(* Logix 5000 project; controller elevatorPart5 vendor 1 type 14 code 106 rev 28.11; software revision 28.03 *)

TASK MainTask (continuous, watchdog 500 ms) : MainProgram

MODULES
   Local : vendor 1 type 14 code 106 (Compact 0, rev 28.11)
       : vendor 1 type 7 code 77 (Compact 2, rev 3.1, Input RPI 20 ms)
       : 1769-IQ16 (Compact 3, rev 1.1, Input RPI 20 ms)
       : vendor 1 type 7 code 72 (Compact 5, rev 2.1, Output RPI 20 ms)
       : vendor 1 type 7 code 72 (Compact 4, rev 2.1, Output RPI 20 ms)
END_MODULES

ADD_ON_INSTRUCTION serviceDoor   (* revision 1.0 *)
VAR_OUTPUT
   serviceDoor : BOOL; {visible}
   doorOpen : BOOL; {visible}
   doorClosed : BOOL; {access Read Only, visible}
END_VAR
VAR_IN_OUT
   doorOpenSensor : BOOL; {required}
   doorClosedSensor : BOOL; {required}
END_VAR
VAR_OUTPUT
   doorControl : SINT; {access Read Only, visible}
END_VAR
VAR_IN_OUT
   pbOpenLyft : BOOL; {required}
   pbCloseLyft : BOOL; {required}
END_VAR
VAR
   doorOpenTimer : TIMER := (PRE := 5000); {access None}
   doorOpenTran : BOOL; {access None}
   activate : BOOL; {access None}
   lightOn : BOOL; {access None}
END_VAR

ROUTINE Logic   (* ladder *)
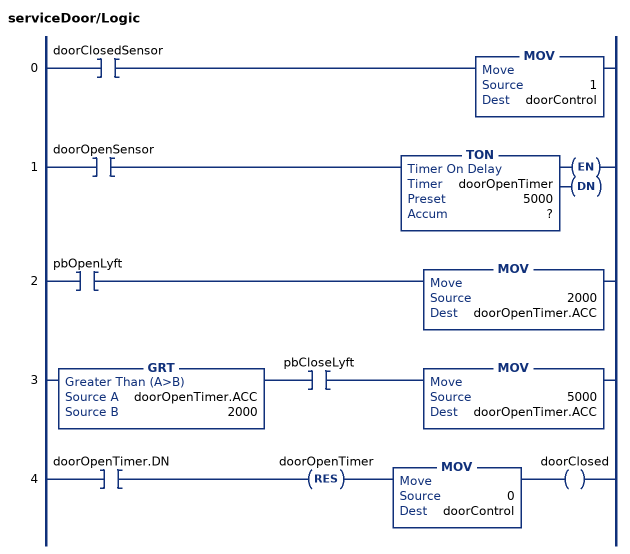
   0: XIC(doorClosedSensor)MOV(1,doorControl);
   1: XIC(doorOpenSensor)TON(doorOpenTimer,?,?);
   2: XIC(pbOpenLyft)MOV(2000,doorOpenTimer.ACC);
   3: GRT(doorOpenTimer.ACC,2000)XIC(pbCloseLyft)MOV(5000,doorOpenTimer.ACC);
   4: XIC(doorOpenTimer.DN)RES(doorOpenTimer)MOV(0,doorControl)OTE(doorClosed);
END_ROUTINE
END_ADD_ON_INSTRUCTION

PROGRAM MainProgram   (* main routine MainRoutine *)
VAR
   array : DINT[6];
   bits : DINT := 3855;
   bool : serviceDoor; {access Read Only}
   buttonPressDetection : SINT;
   callAddOn : BOOL;
   clearCount : DINT;
   count : DINT := 6;
   count2 : DINT;
   CR0 : ALIAS FOR Local:5:O.Data.4;   // Reverse motor's direction
   currentFloor : DINT := 1;
   currentState : DINT := 2;
   currFloorCntr : DINT;
   DCLS : ALIAS FOR Local:3:I.Data.8;   // limit switch; detects if door is closed
   DOLS : ALIAS FOR Local:3:I.Data.9;   // limit switch; detects if door is open
   door_bool : BOOL;
   doorBit : SINT;
   doorClosedSensor : ALIAS FOR DCLS;
   doorClosedSensorBool : BOOL;
   doorOpenSensor : ALIAS FOR DOLS;
   doorOpenSensorBool : BOOL := 1;
   emergency : BOOL;
   emergencyLight : INT;
   FIL1 : ALIAS FOR Local:4:O.Data.11;   // Indicator light; located on the 1st floor
   FIL2 : ALIAS FOR Local:4:O.Data.10;   // Indicator light; located on the 2nd floor
   FIL3 : ALIAS FOR Local:4:O.Data.9;   // Indicator light; located on the 3rd floor
   FIL4 : ALIAS FOR Local:4:O.Data.8;   // Indicator light; located on the 4th floor
   firstFloorBit : DINT;
   floor4_bit : BOOL;
   floorArray : DINT[5];
   floorCntr : COUNTER;
   floorNumIn : DINT;
   floorNumOut : DINT;
   floorSenseCntr : DINT;
   floorSenseRef : ALIAS FOR Local:3:I.Data;
   floorServiceTimer : FBD_TIMER := (PRE := 3000);
   floorServiceTimer_one_shot : BOOL;
   FLS1 : ALIAS FOR Local:3:I.Data.0;   // limit switch; detects if elevator is at 1st floor
   FLS2 : ALIAS FOR Local:3:I.Data.1;   // limit switch; detects if elevator is at 2 nd floor
   FLS3 : ALIAS FOR Local:3:I.Data.2;   // limit switch;detects if elevator is at 3rd floor
   FLS4 : ALIAS FOR Local:3:I.Data.3;   // limit switch; detects if elevator is at 4th floor
   FPB1 : ALIAS FOR Local:2:I.Data.11;   // PB to call elevator; 1 st floor
   FPB2 : ALIAS FOR Local:2:I.Data.10;   // PB to call elevator; 2nd floor
   FPB3 : ALIAS FOR Local:2:I.Data.9;   // PB to call elevator; 3rd floor
   FPB4 : ALIAS FOR Local:2:I.Data.8;   // PB to call elevator; 4th floor
   highSortBit : BOOL := 1;
   highSortValue : BOOL := 1;
   i : DINT := 4;
   IL1 : ALIAS FOR Local:4:O.Data.3;   // Indicator light; floor 1; inside the elvator's panel
   IL2 : ALIAS FOR Local:4:O.Data.2;   // Indicator light; floor 2; inside the elvator's panel
   IL3 : ALIAS FOR Local:4:O.Data.1;   // Indicator light; floor 3; inside the elvator's panel
   IL4 : ALIAS FOR Local:4:O.Data.0;   // Indicator light; floor 4; inside the elvator's panel
   ILC : ALIAS FOR Local:4:O.Data.5;   // Indicator light; if door is closed
   ilc_bit : INT;
   ilc_bool : BOOL;
   ILE5 : ALIAS FOR Local:4:O.Data.6;   // Indicator light; emergency stop button
   ILO : ALIAS FOR Local:4:O.Data.4;   // Indicator light; if door is open
   ILTS0 : ALIAS FOR Local:4:O.Data.14;   // Indicator light; toggle switch 0
   ILTS1 : ALIAS FOR Local:4:O.Data.13;   // Indicator light; toggle switch 1
   ILTS2 : ALIAS FOR Local:4:O.Data.12;   // Indicator light; toggle switch 2
   inFloorBits : INT;
   inPbBool : BOOL;
   inPbCntr : DINT := 1;
   inPbFloor : ALIAS FOR Local:2:I.Data;
   inside_button_4 : BOOL;
   insideLight : DINT;
   j : DINT;
   lightRef : ALIAS FOR Local:4:O.Data;
   lowSortBit : BOOL := 1;
   lowSortValue : BOOL := 1;
   M0 : ALIAS FOR Local:5:O.Data.0;   // Motor for elevator
   maxElementCntr : DINT := 4;
   maxElementValue : SINT := 4;
   min : DINT;
   minElementCntr : SINT := 4;
   minElementValue : SINT;
   motor_bit : BOOL;
   nextFloor : DINT;
   nextFloorCntr : SINT;
   nextState : DINT := 2;
   numFloors : SINT;
   numFloorsCntr : SINT := 4;
   numTempFloors : SINT;
   one_shot : BOOL;
   one_shot_in : BOOL;
   one_shot_out : BOOL;
   outFloorBits : INT;
   outPbBool : BOOL;
   outPbCntr : INT := 10;
   outPbFloor : ALIAS FOR Local:2:I.Data;
   outsideLight : DINT;
   PB1 : ALIAS FOR Local:2:I.Data.3;   // push button 1st floor
   PB2 : ALIAS FOR Local:2:I.Data.2;   // push button 2nd floor
   PB3 : ALIAS FOR Local:2:I.Data.1;   // push button 3rd floor
   PB4 : ALIAS FOR Local:2:I.Data.0;   // push button 4th floor
   PBC : ALIAS FOR Local:2:I.Data.5;   // push button to close door
   PBE5 : ALIAS FOR Local:2:I.Data.6;   // push button to emergency stop lift
   PBO : ALIAS FOR Local:2:I.Data.4;   // push button to open door
   prevFloor : SINT;
   reverse_bit : BOOL;
   serviceDoor : serviceDoor;
   serviceDoorBool : SINT;
   shiftCount : DINT;
   SOL0 : ALIAS FOR Local:5:O.Data.2;   // Solenoid for pneumatic piston; open/close the door
   sorting : DINT;
   sortingCntr : DINT;
   START : ALIAS FOR Local:2:I.Data.14;   // NO start button
   start_bit : BOOL;
   STOP : ALIAS FOR Local:2:I.Data.15;   // NC stop button
   stop_bit : BOOL := 1;
   temp : DINT;
   tempArray : SINT[5];
   tempFloor : SINT := 4;
   testTimer : TIMER := (PRE := 5000, ACC := 8260);
   testValue : BOOL := 1;
   timer1 : TIMER;
   timer1Preset : DINT;
   TS0 : ALIAS FOR Local:3:I.Data.12;   // Toggle switch 0
   TS1 : ALIAS FOR Local:3:I.Data.11;   // Toggle switch 1
   TS2 : ALIAS FOR Local:3:I.Data.10;   // Toggle switch 2
   zeroFloorCntr : DINT := 4;
END_VAR

ROUTINE burnData   (* structured text *)
   
   
   /******************************************************
   * Description: This SBR is to delete all the data
   * 			   at the begining of the lyft's operation
   *
   * Author: Iakov Umrikhin
   * Date created: 06.04.2022
   *******************************************************/
   SBR();
   
   	firstFloorBit := 1;
   
   	currentState := 0;
   	nextState := 0;
   
   	floorSenseRef := 0;
   	floorSenseCntr := 0;
   
       currentFloor := 1;
   	currFloorCntr := 0;
   
   	nextFloor := 0;
   	nextFloorCntr := 0;
   
   	inFloorBits := 0;
   	outFloorBits := 0;
   
   	one_shot := 0;
   
   	emergencyLight := 0;
   	door_bool := 0;
   
   	floorServiceTimer.Reset := 1;
   	zeroFloorCntr := 0;
   
   	prevFloor := 0;
   
   	JSR(clearArray);
   
   	nextState := 0;
   
   
END_ROUTINE

ROUTINE clearArray   (* structured text *)
   
   
   /******************************************************
   * Description:
   *
   *
   * Author: Iakov Umrikhin
   * Date created: March - April, 2022
   *******************************************************/
   
   SBR();
   
   	FOR clearCount := 0 to 4 DO
   		floorArray[clearCount] := 0;
   	END_FOR;
   	clearCount := 0;
   
END_ROUTINE

ROUTINE countFloors   (* structured text *)
   
   
   SBR();
   
   	FOR numFloorsCntr := 0 to 3 DO
   
   		IF floorArray[numFloorsCntr] > 0 THEN
   			numFloors := numFloors + 1;
   		END_IF;
   
   	END_FOR;
   
   	nextFloorCntr := numFloors;
   
   	numFloors := 0;
END_ROUTINE

ROUTINE countFloorsTemp   (* structured text *)
   
   
   SBR();
   
   	FOR numFloorsCntr := 0 to 3 DO
   
   		IF tempArray[numFloorsCntr] > 0 THEN
   			numFloors := numFloors + 1;
   		END_IF;
   
   	END_FOR;
   
   	numTempFloors := numFloors;
   
   	numFloors := 0;
END_ROUTINE

ROUTINE downDirectionSort   (* structured text *)
   SBR();
   
   
   	JSR(highSort);
   	JSR(countFloors);
   
   	FOR i := 0 to (nextFloorCntr - 1) DO
   		IF floorArray[i] > currentFloor THEN
   			tempArray[i] := floorArray[0];
   			JSR(elementShiftLeft);
   			floorArray[nextFloorCntr - i - 1] := 0;
   		END_IF;
   	END_FOR;
   
   	JSR(countFloorsTemp);
   	JSR(countFloors);
   
   	FOR j := 0 TO (numTempFloors - 1) DO
   		floorArray[j + nextFloorCntr] := tempArray[j];
   	END_FOR;
END_ROUTINE

ROUTINE elementShiftLeft   (* structured text *)
   /******************************************************
   * Description:
   *
   *
   * Author: Iakov Umrikhin
   * Date created: March - April, 2022
   *******************************************************/
   
   SBR();
   
   	FOR shiftCount := 0 to 3 DO
   
   		floorArray[shiftCount] := floorArray[shiftCount + 1];
   
   	END_FOR;
   
   	shiftCount := 0;
   
END_ROUTINE

ROUTINE elevatorMain   (* structured text *)
   
   /******************************************************
   * Description:
   *
   *
   * Author: Iakov Umrikhin
   * Date created: 06.04.2022
   *******************************************************/
   
   // Part 5: Emergency button
   
   // initialise START bit
   start_bit := START;
   stop_bit := STOP;
   emergency := PBE5;
   
   // initiallise timer
   floorServiceTimer.PRE := 3000;
   floorServiceTimer.ACC := 0;
   
   (***********************
    * NOTES
    * outPbFloor : 11 -> FPB1R
    				 8 -> FPB4
      inPbFloor: 	3 -> PB1
      		b		0 -> PB4
   	*)
   
   IF S:FS THEN
   
   	JSR(burnData);
   
   END_IF;
   
   // change an intermediate state
   IF currentState <> nextState THEN
       currentState := nextState;
   END_IF;
   
   
   // main states
   // state 0: launch the system:
   
   IF (currentState = 0 AND nextState = 0) THEN
   
   	IF start_bit THEN
   		nextState := 1;
   	END_IF;
   
   END_IF;
   
   						// state 1
   
   IF (currentState = 1 AND nextState = 1) THEN
   
     	IF floorSenseRef.0 THEN
   
   		// move to a next state
   	    nextState := 2;
       END_IF;
   
   	outFloorBits.11 := 1;
   
   	// turn the motor on
   
   	// to make sure that the lyft doesn't burst through the roof
   	// reverse its motion
   
   END_IF;
   
   // transition from State 1 to 2
   IF (currentState = 1 AND nextState = 2) THEN
   
   	IF firstFloorBit = 1 THEN
   		outFloorBits := 0;
   		firstFloorBit := 0;
   	END_IF;
   
   	IF floorArray[currFloorCntr] = 0  OR nextFloorCntr = -1 THEN
   
   		JSR(clearArray); // subroutine
   		outFloorBits := 0;
   		inFloorBits := 0;
   
   		JSR(countFloors);
   	END_IF;
   
   	zeroFloorCntr := 0;
   
   END_IF;
   
   						// state 2: wait for a call
   
   IF (currentState = 2 AND nextState = 2) THEN
   
   	// move to a next state
   	IF floorServiceTimer.DN THEN
   
   		IF (serviceDoorBool = 1) THEN
   
   			nextState := 4;
   
   		ELSE
   
   			nextState := 3;
   
   		END_IF;
   
   	END_IF;
   
   	// increase the currFloorCntr only if there is a floor
   	// to move to
   	floorServiceTimer.Reset := 0;
   	// maybe you could remove bits.[N] from the IF
   	// statement. Should it work, then the code looks simpler
   	// check if the outside panel button is pressed
   
   	outPbBool [:=] outPbFloor.11 OR outPbFloor.10 OR outPbFloor.9 OR outPbFloor.8;
   	inPbBool [:=] inPbFloor.3 OR inPbFloor.2 OR inPbFloor.1 OR inPbFloor.0;
   
   	floorNumOut := bits AND outPbFloor;
   	floorNumIn := bits AND inPbFloor;
   
   	IF outPbBool AND NOT one_shot_out THEN
   		// enable the floorServiceTimer
   
   		floorNumOut := 2048 / floorNumOut;
   
   		CASE floorNumOut OF
   			1:
   				floorNumOut := 1;
   			2:
   				floorNumOut := 2;
   			4:
   				floorNumOut := 3;
   			8:
   				floorNumOut := 4;
   		END_CASE;
   
   		outPbCntr := 12 - floorNumOut;
   
   		outFloorBits.[outPbCntr] := 1;
   		floorArray[nextFloorCntr] := floorNumOut;
   
   		// reset the floorServiceTimer
   		floorServiceTimer.Reset := 1;
   
   		nextFloorCntr := nextFloorCntr + 1;
   		buttonPressDetection := 1;
   	END_IF;
   
   	one_shot_out := outPbBool;
   
   
   	// check if the inside panel button is pressed
   	IF inPbBool AND NOT one_shot_in THEN
   
   		floorNumIn := 8 / floorNumIn;
   
   		CASE floorNumIn OF
   			1:
   				floorNumIn := 1;
   			2:
   				floorNumIn := 2;
   			4:
   				floorNumIn := 3;
   			8:
   				floorNumIn := 4;
   		END_CASE;
   
   		inPbCntr := 4 - floorNumIn;
   
   		inFloorBits.[inPbCntr] := 1;
   		floorArray[nextFloorCntr] := floorNumIn;
   
   		// reset the floorServiceTimer
   		floorServiceTimer.Reset := 1;
   
   		nextFloorCntr := nextFloorCntr + 1;
   		buttonPressDetection := 1;
   	END_IF;
   
   	one_shot_in := inPbBool;
   
   	IF nextFloorCntr > 4 THEN
   
   		nextFloorCntr := 0;
   		JSR(clearArray);
   
   		outFloorBits := 0;
   		inFloorBits := 0;
   	END_IF;
   
   	IF floorArray[currFloorCntr] >= 1 AND NOT floorServiceTimer_one_shot THEN
   		floorServiceTimer.TimerEnable := 1;
   	END_IF;
   
   	TONR(floorServiceTimer);
   
   	floorServiceTimer_one_shot [:=] floorServiceTimer.EN;
   
   END_IF;
   
   // transition from State 2 to 4
   IF (currentState = 2 AND nextState = 4) THEN
   		floorServiceTimer.DN := 0;
   		floorServiceTimer.Reset := 1;
   		floorServiceTimer.TimerEnable := 0;
   		serviceDoorBool := 0;
   END_IF;
   
   // transition from State 2 to 3; sort the list of floors
   IF (currentState = 2 AND nextState = 3) THEN
   
   	// desable the floorServiceTimer
   	// reset the floorServiceTimer
   	floorServiceTimer.DN := 0;
   	floorServiceTimer.Reset := 1;
   	floorServiceTimer.TimerEnable := 0;
   
   
   	JSR(countFloors);
   
   (*			MULTIPLE-CALLS ALGORITHMS. Start			*)
   
   	IF currentFloor = 1 THEN
   		JSR(lowSort);
   		JSR(maxElement);
   	END_IF;
   
   	IF currentFloor = 4 THEN
   		maxElementValue := 0;
   		JSR(highSort);
   		JSR(minElement);
   		prevFloor := 4;
   	END_IF;
   
   //	IF currentFloor = 3 AND prevFloor = 4 THEN
   	IF prevFloor = 4 THEN
   
   		JSR(downDirectionSort);
   
   		// floor swap
   		IF floorArray[currFloorCntr] = 4 THEN
   			tempFloor := floorArray[currFloorCntr];
   			JSR(elementShiftLeft);
   			floorArray[nextFloorCntr-1] := tempFloor;
   		END_IF;
   		// end
   		prevFloor := 0;
   	END_IF;
   
   	IF (maxElementValue = currentFloor) AND (currentFloor <> 4) THEN
   
   		JSR(maxElement);
   
   		IF maxElementValue > currentFloor THEN
   			JSR(highSort);
   		ELSE
   			maxElementValue := 0;
   			JSR(highSort);
   			JSR(minElement);
   		END_IF;
   
   	END_IF;
   
   	IF (minElementValue = currentFloor) THEN
   
   		minElementValue := 0;
   		JSR(lowSort);
   		JSR(maxElement);
   
   	END_IF;
   
   (*			MULTIPLE-CALLS ALGORITHMS. End			*)
   
   	// floor repeats or it is zero; shift by one to the left
   	// if there are more than 4 zeros in the array then the array is empty
   	WHILE (floorArray[currFloorCntr] = floorArray[currFloorCntr + 1] OR floorArray[currFloorCntr] = 0) AND (zeroFloorCntr <> 4) DO
   
   		IF (floorArray[currFloorCntr] = 0) THEN
   			zeroFloorCntr := zeroFloorCntr + 1;
   		END_IF;
   
   		JSR(elementShiftLeft);
   
   	END_WHILE;
   
   	// check if the array's element is zero
   	// act accordingly
   	IF floorArray[currFloorCntr] = 0 THEN
   
   		JSR(elementShiftLeft);
   
   	END_IF;
   
   	// calculate which floor's sensor to stop at
   	floorSenseCntr := floorArray[currFloorCntr] - 1;
   
   	JSR(countFloors);
   END_IF;
   
   						// state 3: move to a floor
   
   IF (currentState = 3 AND nextState = 3) THEN
   
   	// check if the called floor's sensor is on
   	IF floorSenseRef.[floorSenseCntr] THEN
   
   		nextState := 4;
   	END_IF;
   
   
   	// turn the motor on
   
   	(* if the next floor is lower than the current floor
   	   then reverse the direction of the lyft *)
   
   END_IF;
   
   // transition from state 3 to state 4;
   IF (currentState = 3 AND nextState = 4) THEN
   
   	currentFloor := floorArray[currFloorCntr];
   
   	outFloorBits.[12 - currentFloor] := 0;
   	inFloorBits.[4 - currentFloor] := 0;
   
   	serviceDoorBool := 1;
   
   END_IF;
   						// state 4: stop the motion; return to State 2
   
   IF (currentState = 4 AND nextState = 4) THEN
   
   	IF (serviceDoorBool = 1) THEN
   		nextState := 2;	// wait for 3 seconds to service a floor
   	END_IF;
   
   	IF (serviceDoorBool <> 1) THEN
   		JSR(timerService);
   	END_IF;
   
   	outPbBool [:=] outPbFloor.11 OR outPbFloor.10 OR outPbFloor.9 OR outPbFloor.8;
   	inPbBool [:=] inPbFloor.3 OR inPbFloor.2 OR inPbFloor.1 OR inPbFloor.0;
   
   	floorNumOut := bits AND outPbFloor;
   	floorNumIn := bits AND inPbFloor;
   
   	IF outPbBool AND NOT one_shot_out THEN
   		// enable the floorServiceTimer
   
   		floorNumOut := 2048 / floorNumOut;
   
   		CASE floorNumOut OF
   			1:
   				floorNumOut := 1;
   			2:
   				floorNumOut := 2;
   			4:
   				floorNumOut := 3;
   			8:
   				floorNumOut := 4;
   		END_CASE;
   
   		outPbCntr := 12 - floorNumOut;
   
   		outFloorBits.[outPbCntr] := 1;
   		floorArray[nextFloorCntr] := floorNumOut;
   
   		// reset the floorServiceTimer
   		floorServiceTimer.Reset := 1;
   
   		nextFloorCntr := nextFloorCntr + 1;
   		buttonPressDetection := 1;
   	END_IF;
   
   	one_shot_out := outPbBool;
   
   
   	// check if the inside panel button is pressed
   	IF inPbBool AND NOT one_shot_in THEN
   
   		floorNumIn := 8 / floorNumIn;
   
   		CASE floorNumIn OF
   			1:
   				floorNumIn := 1;
   			2:
   				floorNumIn := 2;
   			4:
   				floorNumIn := 3;
   			8:
   				floorNumIn := 4;
   		END_CASE;
   
   		inPbCntr := 4 - floorNumIn;
   
   		inFloorBits.[inPbCntr] := 1;
   		floorArray[nextFloorCntr] := floorNumIn;
   
   		// reset the floorServiceTimer
   		floorServiceTimer.Reset := 1;
   
   		nextFloorCntr := nextFloorCntr + 1;
   		buttonPressDetection := 1;
   	END_IF;
   
   	one_shot_in := inPbBool;
   
   	IF nextFloorCntr > 4 THEN
   
   		nextFloorCntr := 0;
   		JSR(clearArray);
   
   		outFloorBits := 0;
   		inFloorBits := 0;
   	END_IF;
   
   END_IF;
   
   IF (currentState = 4 AND nextState = 2) THEN
   
   	IF (serviceDoorBool <> 1) THEN
   
   		JSR(elementShiftLeft);
   
   		JSR(countFloors);
   
   		// floor repeats or it is zero; shift by one to the left
   		// if there are more than 4 zeros in the array then the array is empty
   		WHILE (floorArray[currFloorCntr] = floorArray[currFloorCntr + 1] OR floorArray[currFloorCntr] = 0) AND (zeroFloorCntr <> 4) DO
   
   			IF (floorArray[currFloorCntr] = 0) THEN
   				zeroFloorCntr := zeroFloorCntr + 1;
   			END_IF;
   
   			JSR(elementShiftLeft);
   
   		END_WHILE;
   
   		IF (buttonPressDetection <> 1) THEN
   			floorArray[nextFloorCntr] := 0;
   			nextFloorCntr := nextFloorCntr - 1;
   			JSR(countFloors);
   		END_IF;
   
   		buttonPressDetection := 0;
   
   	END_IF;
   END_IF;
   						// EMERGENCY STATE
   IF emergency THEN
   	nextState := 5;
   END_IF;
   
   
   IF (currentState = 5 AND nextState = 5) THEN
   
   	emergencyLight := 64; // 5th bit
   
   	// if one of the sensors is active
   	// the lyft is on one of the floors
   	IF (floorSenseRef.[floorSenseCntr]) THEN
   		door_bool [:=] 1;
   	END_IF;
   
   	// if the emergency occurs between floors;
   	// only possible, when neither of sensors is on
   
   	IF start_bit THEN
   		nextState := 0;
   	END_IF;
   
   END_IF;
   
   // Transition from State 5 to 2; clear all data
   IF (currentState = 5 AND nextState = 0) THEN
   
   	JSR(burnData);
   
   END_IF;
   
   // if stop pressed clear everything and
   // return to state 1
   IF NOT stop_bit THEN
   
   	JSR(burnData);
   
   END_IF;
   
   (* OUTPUT SECTION *)
   
   //
   
   // output for the outside panel lights
   lightRef := outFloorBits OR inFloorBits OR ilc_bit OR emergencyLight;
   
   // elevator's door bit
   SOL0 := door_bool;
   
   
   // output for motor's bits
   M0 [:=] (currentState = 1 AND nextState = 1) OR (currentState = 3 AND nextState = 3);
   CR0 [:=] ((currentState = 1 AND nextState = 1) AND NOT floorSenseRef.0) OR ((currentState = 3 AND nextState = 3) AND (floorArray[currFloorCntr] < currentFloor));
   
END_ROUTINE

ROUTINE highSort   (* structured text *)
// Sorting an array from hight to low values
   /******************************************************
   * Description:
   *
   *
   * Author: Iakov Umrikhin
   * Date created: March - April, 2022
   *******************************************************/
   
   SBR();
   
       FOR i:= 1 to 3 DO
   		min := floorArray[i];
   		j := i - 1;
           WHILE j >= 0 AND floorArray[j] < min DO
   			floorArray[j + 1] := floorArray[j];
   			j := j - 1;
   		END_WHILE;
   		floorArray[j + 1] := min;
   	END_FOR;
   	j := 0;
END_ROUTINE

ROUTINE lowSort   (* structured text *)
// Sorting an array from low to high values
   /******************************************************
   * Description:
   *
   *
   * Author: Iakov Umrikhin
   * Date created: March - April, 2022
   *******************************************************/
   
   SBR();
   
       FOR i:= 1 to 3 DO
   		min := floorArray[i];
   		j := i - 1;
           WHILE j >= 0 AND floorArray[j] > min DO
   			floorArray[j + 1] := floorArray[j];
   			j := j - 1;
   		END_WHILE;
   		floorArray[j + 1] := min;
   	END_FOR;
   
   	j := 0;
END_ROUTINE

ROUTINE MainRoutine   (* ladder *)
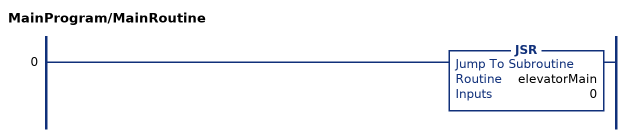
   0: JSR(elevatorMain,0);
END_ROUTINE

ROUTINE maxElement   (* structured text *)
   SBR();
   
   	maxElementValue := 1;
   
   	FOR maxElementCntr := 0 TO 3 DO
   
   		IF (floorArray[maxElementCntr] > maxElementValue AND floorArray[maxElementCntr] <> 0) THEN
   			maxElementValue := floorArray[maxElementCntr];
   		END_IF;
   
   	END_FOR;
END_ROUTINE

ROUTINE minElement   (* structured text *)
   SBR();
   
   	minElementValue := 4;
   
   	FOR minElementCntr := 0 TO 3 DO
   
   		IF (floorArray[minElementCntr] < minElementValue AND floorArray[minElementCntr] <> 0) THEN
   			minElementValue := floorArray[minElementCntr];
   		END_IF;
   
   	END_FOR;
END_ROUTINE

ROUTINE timerService   (* ladder *)
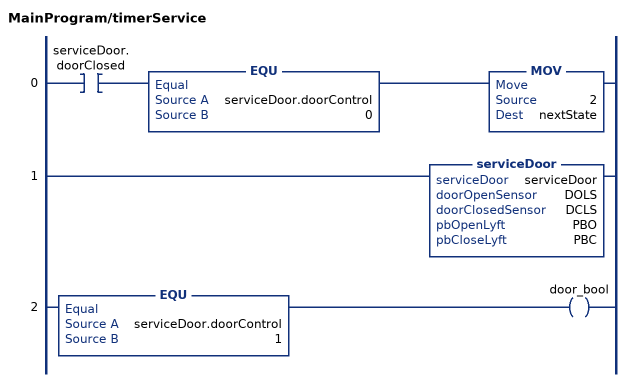
   0: XIC(serviceDoor.doorClosed)EQU(serviceDoor.doorControl,0)MOV(2,nextState);
   1: serviceDoor(serviceDoor,DOLS,DCLS,PBO,PBC);
   2: EQU(serviceDoor.doorControl,1)OTE(door_bool);
END_ROUTINE
END_PROGRAM
